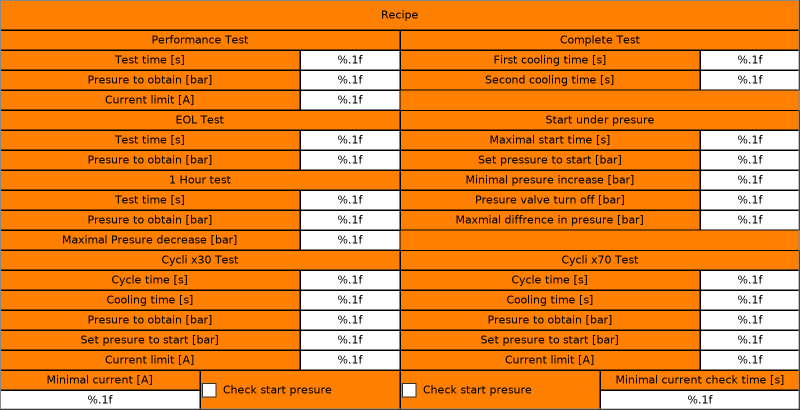
VISUALIZATION vRecipe  // 800x410
VAR_IN_OUT
	fbChamber 	: fbChamber;
	stChamberTestParams	: stTestParams;
END_VAR
    Rectangle (200,370 200x40)
    Rectangle (0,0 800x30), "Recipe"
    Rectangle (0,30 400x20), "Performance Test"
    Rectangle (0,50 300x20), "Test time [s]"
    Rectangle (0,70 300x20), "Presure to obtain [bar]"
    Rectangle (0,90 300x20), "Current limit [A]"
    Rectangle (0,110 400x20), "EOL Test"
    Rectangle (0,130 300x20), "Test time [s]"
    Rectangle (0,150 300x20), "Presure to obtain [bar]"
    Rectangle (0,190 300x20), "Test time [s]"
    Rectangle (0,170 400x20), "1 Hour test"
    Rectangle (0,210 300x20), "Presure to obtain [bar]"
    Rectangle (0,230 300x20), "Maximal Presure decrease [bar]"
    Rectangle (400,50 300x20), "First cooling time [s]"
    Rectangle (400,30 400x20), "Complete Test"
    Rectangle (400,70 300x20), "Second cooling time [s]"
    Rectangle (400,110 400x20), "Start under presure"
    Rectangle (400,130 300x20), "Maximal start time [s]"
    Rectangle (400,150 300x20), "Set pressure to start [bar]"
    Rectangle (400,170 300x20), "Minimal presure increase [bar]"
    Rectangle (400,210 300x20), "Maxmial diffrence in presure [bar]"
    Rectangle (400,190 300x20), "Presure valve turn off [bar]"
    Rectangle (400,250 400x20), "Cycli x70 Test"
    Rectangle (0,250 400x20), "Cycli x30 Test"
    Rectangle (0,350 300x20), "Current limit [A]"
    Rectangle (0,270 300x20), "Cycle time [s]"
    Rectangle (0,290 300x20), "Cooling time [s]"
    Rectangle (0,310 300x20), "Presure to obtain [bar]"
    Rectangle (0,330 300x20), "Set presure to start [bar]"
    Checkbox (200,375 200x30), "Check start presure", variable: stChamberTestParams.bCheckStartPresureCycle30
    Rectangle (400,370 200x40)
    Rectangle (400,350 300x20), "Current limit [A]"
    Rectangle (400,270 300x20), "Cycle time [s]"
    Rectangle (400,290 300x20), "Cooling time [s]"
    Rectangle (400,310 300x20), "Presure to obtain [bar]"
    Rectangle (400,330 300x20), "Set presure to start [bar]"
    Checkbox (400,375 200x30), "Check start presure", variable: stChamberTestParams.bCheckStartPresureCycle70
    Rectangle (300,50 100x20), "%.1f", text variable: stChamberTestParams.rTest300SecTime
        OnMouseClick: write the text variable via Default, min 0, max 10000000
    Rectangle (300,70 100x20), "%.1f", text variable: stChamberTestParams.rPresureToObtainPerformanceTest
        OnMouseClick: write the text variable via Default, min 0, max 10
    Rectangle (300,90 100x20), "%.1f", text variable: stChamberTestParams.rCurrentLimitPerformacneTest
        OnMouseClick: write the text variable via Default, min 1, max 20
    Rectangle (300,190 100x20), "%.1f", text variable: stChamberTestParams.rTestHourTime
        OnMouseClick: write the text variable via Default, min 0, max 10000000
    Rectangle (300,210 100x20), "%.1f", text variable: stChamberTestParams.rPressureToObtainHourTest
        OnMouseClick: write the text variable via Default, min 0, max 10
    Rectangle (300,230 100x20), "%.1f", text variable: stChamberTestParams.rTestHourPressureMaximalTolerance
        OnMouseClick: write the text variable via Default, min 0, max 10
    Rectangle (700,50 100x20), "%.1f", text variable: stChamberTestParams.rTestCoolingTimeFullStepI
        OnMouseClick: write the text variable via Default, min 0, max 10000000
    Rectangle (700,70 100x20), "%.1f", text variable: stChamberTestParams.rTestCoolingTimeFullStepII
        OnMouseClick: write the text variable via Default, min 0, max 10000000
    Rectangle (700,150 100x20), "%.1f", text variable: stChamberTestParams.rTestUnderPresureSetPresure
        OnMouseClick: write the text variable via Default, min 0, max 10
    Rectangle (700,130 100x20), "%.1f", text variable: stChamberTestParams.rTestUnderPresureTime
        OnMouseClick: write the text variable via Default, min 0, max 10000000
    Rectangle (700,170 100x20), "%.1f", text variable: stChamberTestParams.rTestUnderPresureMinimalIncrease
        OnMouseClick: write the text variable via Default, min 0, max 10
    Rectangle (700,210 100x20), "%.1f", text variable: stChamberTestParams.rTestUnderPresureStartTolerance
        OnMouseClick: write the text variable via Default, min 0, max 10
    Rectangle (700,190 100x20), "%.1f", text variable: stChamberTestParams.rTestUnderPresureCloseTolerance
        OnMouseClick: write the text variable via Default, min 0, max 10
    Rectangle (300,350 100x20), "%.1f", text variable: stChamberTestParams.rCurrentLimitCycle30
        OnMouseClick: write the text variable via Default, min 0, max 10
    Rectangle (300,310 100x20), "%.1f", text variable: stChamberTestParams.rPresureToObtainCycle30Test
        OnMouseClick: write the text variable via Default, min 0, max 10
    Rectangle (300,330 100x20), "%.1f", text variable: stChamberTestParams.rStartPresureCycle30Test
        OnMouseClick: write the text variable via Default, min 0, max 10
    Rectangle (300,270 100x20), "%.1f", text variable: stChamberTestParams.rTestCycle30LimitTime
        OnMouseClick: write the text variable via Default, min 0, max 10000000
    Rectangle (300,290 100x20), "%.1f", text variable: stChamberTestParams.rTestCycle30CoolingTime
        OnMouseClick: write the text variable via Default, min 0, max 10000000
    Rectangle (700,350 100x20), "%.1f", text variable: stChamberTestParams.rCurrentLimitCycle70
        OnMouseClick: write the text variable via Default, min 0, max 10
    Rectangle (700,310 100x20), "%.1f", text variable: stChamberTestParams.rPresureToObtainCycle70Test
        OnMouseClick: write the text variable via Default, min 0, max 10
    Rectangle (700,330 100x20), "%.1f", text variable: stChamberTestParams.rStartPresureCycle70Test
        OnMouseClick: write the text variable via Default, min 0, max 10
    Rectangle (700,270 100x20), "%.1f", text variable: stChamberTestParams.rTestCycle70LimitTime
        OnMouseClick: write the text variable via Default, min 0, max 10000000
    Rectangle (700,290 100x20), "%.1f", text variable: stChamberTestParams.rTestCycle70CoolingTime
        OnMouseClick: write the text variable via Default, min 0, max 10000000
    Rectangle (300,130 100x20), "%.1f", text variable: stChamberTestParams.rTestEolLimitTime
        OnMouseClick: write the text variable via Default, min 0, max 10000000
    Rectangle (300,150 100x20), "%.1f", text variable: stChamberTestParams.rPresureToObtainEOLTest
        OnMouseClick: write the text variable via Default, min 0, max 10
    Rectangle (0,370 200x20), "Minimal current [A]"
    Rectangle (0,390 200x20), "%.1f", text variable: stChamberTestParams.rMinimalCurrentLimit
        OnMouseClick: write the text variable via Default, min 0, max 10
    Rectangle (600,370 200x20), "Minimal current check time [s]"
    Rectangle (600,390 200x20), "%.1f", text variable: stChamberTestParams.rMinimalCurrentCheckDelay
        OnMouseClick: write the text variable via Default, min 0, max 10
END_VISUALIZATION

(* stored: Version 1.1.0.1, ProductVersion 3.1.4024.12
   Visu vRecipe: Id {323db5ed-a182-49d7-86c7-3bc24bbe371d} *)
